PROGRAM prg_Parking
VAR
	Sensor1, Sensor2    AT	 	%I*		:BOOL;
	bBinnen               : BOOL;
 	Slagboom       		AT 		%Q* 	:BOOL;
	Roodlicht			AT		%Q*		:BOOL;
	Groenlicht			AT		%Q*		:BOOL;
	AantalAutos			AT		%Q*		:INT;
	AutoTeller: CTUD;
	BinnenRising: R_TRIG;
	BuitenRising: R_TRIG;
	BinnenFalling: F_TRIG;
	BuitenFalling: F_TRIG;
END_VAR

BinnenRising(CLK:= Sensor1);
BuitenRising(CLK:= Sensor2);
BinnenFalling(CLK:= Sensor1);
BuitenFalling(CLK:= Sensor2);


IF BinnenRising.Q THEN
	bBinnen:=TRUE;
ELSIF BuitenRising.Q THEN
	bBinnen:=FALSE;
END_IF

Slagboom := Sensor1 OR Sensor2;

AutoTeller(
	CU:= (bBinnen AND BuitenFalling.Q), 
	CD:= (NOT(bBinnen) AND BinnenFalling.Q), 
	LOAD:= 0, 
	PV:= 10, //10 autos 
	);
IF AutoTeller.CV >= AutoTeller.PV THEN
	Roodlicht:=TRUE;
	Groenlicht:=FALSE;
ELSIF AutoTeller.CV < AutoTeller.PV THEN
	Groenlicht:=TRUE;
	Roodlicht:=FALSE;
END_IF

AantalAutos :=  REAL_TO_INT(AutoTeller.CV)*32767 / 10;//Voor tellerstand aan de inkom van de parkeergarage

END_PROGRAM

(* stored: Version 1.1.0.1, ProductVersion 3.1.4024.15
   POU prg_Parking: Id {9366d75b-1989-4a9f-95de-b8db72f8ada3}, SpecialFunc None *)
